// TIA Portal project "water fill station seq method" (V16)
// Vorlageprojekt für das Buch mit Zielsystem S7-1200

(* hardware
DEVICE "S7-1200-Station_1"  S7-1200 Station
   slot 0: "Baugruppenträger_0"  Rack  V1.0
   slot 1: "PLC_1"  CPU 1211C DC/DC/DC  6ES7 211-1AE40-0XB0  V4.1
*)

// ===== PLC "PLC_1"  CPU 1211C DC/DC/DC =====

VAR_GLOBAL   // PLC tag table "Standard-Variablentabelle"
   "start" AT %I0.0 : Bool;
   "stop" AT %I0.1 : Bool;
   "high" AT %I0.2 : Bool;
   "low" AT %I0.3 : Bool;
   "step" AT %MW100 : Int;
   "fill" AT %Q0.0 : Bool;
   "drain" AT %Q0.1 : Bool;
   "mixer" AT %Q0.2 : Bool;
   "Tag_1" AT %M10.2 : Bool;
   "dis" AT %QW30 : Int;
   "Tag_2" AT %M10.3 : Bool;
   "Tag_3" AT %M10.1 : Bool;
   "last step" AT %MW102 : Int;
END_VAR

// folder: System blocks/Program resources

DATA_BLOCK "IEC_Timer_0_DB_4"   // DB5
{ S7_Optimized_Access := 'TRUE' }
AUTHOR : Simatic
FAMILY : IEC
NAME : IEC_TMR
VERSION : 1.0
// stored: InstanceOfName IEC_TIMER
"IEC_TIMER"
BEGIN
END_DATA_BLOCK

// folder: (top level)

FUNCTION "MHJ-PLC-Lab-Function-S71200" : Void   // FC9000, SCL
{ S7_Optimized_Access := 'TRUE' }
VERSION : 0.1
   VAR_TEMP
      rdTimeReturn : Int;
      outputTime : DTL;
      SyncVal : Byte;
      forVal : Int;
      forVal_2 : Int;
      Value : Byte;
   END_VAR
   VAR CONSTANT
      CompVal : Byte := 16#34;
      Value_01 : Byte := 16#11;
      Value_01_DW : DWord := 16#A165_D992;
      Value_02_DW : DWord := 16#58BE_4401;
   END_VAR
BEGIN

   #Value:=PEEK(area := 16#82,
        dbNumber := 0,
        byteOffset := 511);
   #Value := #Value + 1;

   POKE(area := 16#82,
        dbNumber := 0,
        byteOffset := 511,
        value := #Value);

   POKE(area:=16#81,
        dbNumber:=0,
        byteOffset:=1016,
        value:=#Value_01_DW);
   POKE(area := 16#81,
        dbNumber := 0,
        byteOffset := 1020,
        value := #Value_02_DW);

   POKE(area := 16#81,
        dbNumber := 0,
        byteOffset := 511,
        value := B#16#00);

   FOR #forVal := 0 TO 120 DO
       FOR #forVal_2:=0 TO 10 DO
           #rdTimeReturn:=RD_SYS_T(#outputTime);
           #rdTimeReturn := WR_SYS_T(#outputTime);
           #rdTimeReturn := RD_SYS_T(#outputTime);
           #rdTimeReturn := WR_SYS_T(#outputTime);
       END_FOR;
       #SyncVal:= PEEK(area := 16#81,
                      dbNumber := 0,
                      byteOffset := 511);
       IF #SyncVal = #CompVal THEN
          GOTO M_1;
       END_IF;
   END_FOR;
   RETURN;

   M_1:
   POKE(area := 16#81,
        dbNumber := 0,
        byteOffset := 511,
        value := B#16#0);
END_FUNCTION

ORGANIZATION_BLOCK "Main"   // OB1, LAD, ProgramCycle
TITLE = "Main Program Sweep (Cycle)"
{ S7_Optimized_Access := 'TRUE' }
VERSION : 0.1
   VAR_INPUT
      Initial_Call : Bool;   // Initial call of this OB
      Remanence : Bool;   // =True, if remanent data are available
   END_VAR
   VAR_TEMP   // added for the SCL form of the ladder/FBD networks
      _w1 : Bool;
   END_VAR
BEGIN

REGION Network 1
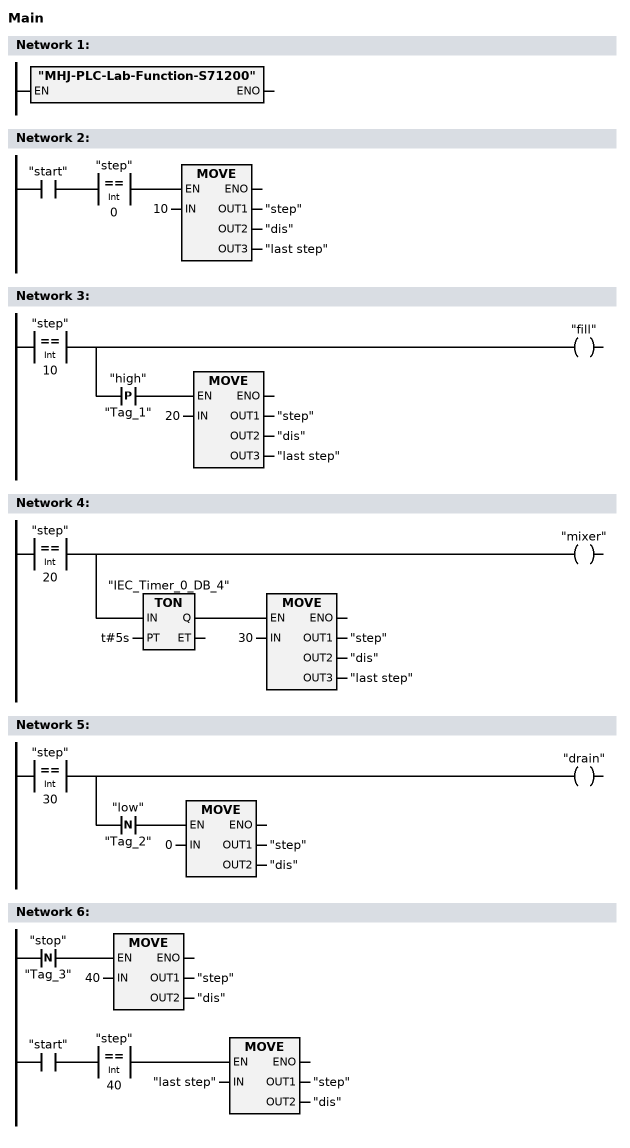
   RUNG wire#powerrail
      "MHJ-PLC-Lab-Function-S71200"()
   END_RUNG
   // the same network as SCL:
   "MHJ-PLC-Lab-Function-S71200"();
END_REGION

REGION Network 2
   RUNG wire#powerrail
      Contact( "start" )
      { S7_Templates := "SrcType := Int" } EQ_Contact(in1 := "step", in2 := 0)
      Move(in := 10, out1 => "step", out2 => "dis", out3 => "last step")
   END_RUNG
   // the same network as SCL:
   IF "start" AND ("step" = 0) THEN
       "step" := 10;
       "dis" := 10;
       "last step" := 10;
   END_IF;
END_REGION

REGION Network 3
   RUNG wire#powerrail
      { S7_Templates := "SrcType := Int" } EQ_Contact(in1 := "step", in2 := 10)
      wire#w1
      Coil( "fill" )
   END_RUNG
   RUNG wire#w1
      P_Contact(operand := "high", bit := "Tag_1")
      Move(in := 20, out1 => "step", out2 => "dis", out3 => "last step")
   END_RUNG
   // the same network as SCL:
   "fill" := "step" = 10;
   #_w1 := "fill" AND "high" AND NOT "Tag_1";   // rising edge of "high"
   "Tag_1" := "high";
   IF #_w1 THEN
       "step" := 20;
       "dis" := 20;
       "last step" := 20;
   END_IF;
END_REGION

REGION Network 4
   "mixer" := "step" = 20;
   "IEC_Timer_0_DB_4".TON(IN := "mixer", PT := t#5s);
   IF "IEC_Timer_0_DB_4".Q THEN
       "step" := 30;
       "dis" := 30;
       "last step" := 30;
   END_IF;
END_REGION

REGION Network 5
   RUNG wire#powerrail
      { S7_Templates := "SrcType := Int" } EQ_Contact(in1 := "step", in2 := 30)
      wire#w1
      Coil( "drain" )
   END_RUNG
   RUNG wire#w1
      N_Contact(operand := "low", bit := "Tag_2")
      Move(in := 0, out1 => "step", out2 => "dis")
   END_RUNG
   // the same network as SCL:
   "drain" := "step" = 30;
   #_w1 := "drain" AND NOT "low" AND "Tag_2";   // falling edge of "low"
   "Tag_2" := "low";
   IF #_w1 THEN
       "step" := 0;
       "dis" := 0;
   END_IF;
END_REGION

REGION Network 6
   RUNG wire#powerrail
      N_Contact(operand := "stop", bit := "Tag_3")
      Move(in := 40, out1 => "step", out2 => "dis")
   END_RUNG
   RUNG wire#powerrail
      Contact( "start" )
      { S7_Templates := "SrcType := Int" } EQ_Contact(in1 := "step", in2 := 40)
      Move(in := "last step", out1 => "step", out2 => "dis")
   END_RUNG
   // the same network as SCL:
   #_w1 := NOT "stop" AND "Tag_3";   // falling edge of "stop"
   "Tag_3" := "stop";
   IF #_w1 THEN
       "step" := 40;
       "dis" := 40;
   END_IF;
   IF "start" AND ("step" = 40) THEN
       "step" := "last step";
       "dis" := "last step";
   END_IF;
END_REGION
END_ORGANIZATION_BLOCK